// Decode a 32-bit value with ZigZag encoding.
FUNCTION F_DecodeZigZag32 : DINT
VAR_INPUT
    nValue : UDINT;
END_VAR

F_DecodeZigZag32 := TO_DINT(SHR(nValue, TO_UDINT(1)) XOR TO_UDINT(-TO_DINT((nValue AND TO_UDINT(1)))));

END_FUNCTION

(* stored: Version 1.1.0.1
   POU F_DecodeZigZag32: Id {e2ea44ff-ba65-4e15-827c-98d6e7575b56}, SpecialFunc None *)
